// TIA Portal V17 export
// export: Created 2026-04-13T11:12:53.8803486Z, ExportSetting WithDefaults, DisplayName Totally Integrated Automation Portal, DisplayVersion V17 Update 4, DisplayName TIA Portal Openness, DisplayVersion V17 Update 4, DisplayName TIA Portal Version Control Interface, DisplayVersion V17, DisplayName SINAMICS Startdrive Advanced, DisplayVersion V17, DisplayName SINAMICS Startdrive G130, G150, S120, S150, SINAMICS MV, S210, DisplayVersion V17, DisplayName SINAMICS Startdrive G110M, G120, G120C, G120D, G120P, G115D, DisplayVersion V17, DisplayName STEP 7 Professional, DisplayVersion V17 Update 4, DisplayName STEP 7 Safety, DisplayVersion V17, DisplayName WinCC Professional, DisplayVersion V17 Update 4
TagTable "SV"
  SV_BD布袋压差高报 : Real  (PLC tag SV.BD布袋压差高报, HMI_连接_1, 1 s)
  SV_BD布袋压差高高报 : Real  (PLC tag SV.BD布袋压差高高报, HMI_连接_1, 1 s)
  SV_JF进风压差高报 : Real  (PLC tag SV.JF进风压差高报, HMI_连接_1, 1 s)
  SV_JF进风压差高高报 : Real  (PLC tag SV.JF进风压差高高报, HMI_连接_1, 1 s)
  SV_TN塔内压力高高报 : Real  (PLC tag SV.TN塔内压力高高报, HMI_连接_1, 1 s)
  SV_GD管道压力高报 : Real  (PLC tag SV.GD管道压力高报, HMI_连接_1, 1 s)
  SV_GD管道压力高高报 : Real  (PLC tag SV.GD管道压力高高报, HMI_连接_1, 1 s)
  SV_GD管道压力设定 : Real  (PLC tag SV.GD管道压力设定, HMI_连接_1, 1 s)
  SV_TN塔内压力低报 : Real  (PLC tag SV.TN塔内压力低报, HMI_连接_1, 1 s)
  SV_TN塔内压力低低报 : Real  (PLC tag SV.TN塔内压力低低报, HMI_连接_1, 1 s)
  SV_XH循风机频率设定 : Real  (PLC tag SV.XH循风机频率设定, HMI_连接_1, 1 s)
  SV_YF引风频率设定 : Real  (PLC tag SV.YF引风频率设定, HMI_连接_1, 1 s)
  SV_JL进料泵频率设定 : Real  (PLC tag SV.JL进料泵频率设定, HMI_连接_1, 1 s)
  SV_JF进风温度设定 : Real  (PLC tag SV.JF进风温度设定, HMI_连接_1, 1 s)
  SV_CF出温异常设定 : Real  (PLC tag SV.CF出温异常设定, HMI_连接_1, 1 s)
  SV_JF进温高报 : Real  (PLC tag SV.JF进温高报, HMI_连接_1, 1 s)
  SV_JF进温高高报 : Real  (PLC tag SV.JF进温高高报, HMI_连接_1, 1 s)
  SV_CF出风温度设定 : Real  (PLC tag SV.CF出风温度设定, HMI_连接_1, 1 s)
  SV_CF出温高报 : Real  (PLC tag SV.CF出温高报, HMI_连接_1, 1 s)
  SV_CF出温高高报 : Real  (PLC tag SV.CF出温高高报, HMI_连接_1, 1 s)
  SV_WQ尾温高报 : Real  (PLC tag SV.WQ尾温高报, HMI_连接_1, 1 s)
  SV_WQ尾温高高报 : Real  (PLC tag SV.WQ尾温高高报, HMI_连接_1, 1 s)
  SV_BD布袋反吹时间 : Real  (PLC tag SV.BD布袋反吹时间, HMI_连接_1, 1 s)
  SV_TW塔外气锤时间 : Real  (PLC tag SV.TW塔外气锤时间, HMI_连接_1, 1 s)
  SV_TN塔内气扫时间 : Real  (PLC tag SV.TN塔内气扫时间, HMI_连接_1, 1 s)
  SV_DQ氮气下限设定 : Real  (PLC tag SV.DQ氮气下限设定, HMI_连接_1, 1 s)
  SV_TN塔内压力高报 : Real  (PLC tag SV.TN塔内压力高报, HMI_连接_1, 1 s)
  SV_JW降温温度设定 : Real  (PLC tag SV.JW降温温度设定, HMI_连接_1, 1 s)
  SV_LS冷水温度写 : Real  (PLC tag SV.LS冷水温度写, HMI_连接_1, 1 s)
  SV_ZT主塔振打间隔 : Real  (PLC tag SV.ZT主塔振打间隔, HMI_连接_1, 1 s)
  SV_TZ通针时间 : Real  (PLC tag SV.TZ通针时间, HMI_连接_1, 1 s)
  SV_PM屏幕编号 : Real  (PLC tag SV.PM屏幕编号, HMI_连接_1, 1 s)
  SV_YH氧含仪高报 : Real  (PLC tag SV.YH氧含仪高报, HMI_连接_1, 1 s)
  SV_JD进氮压力 : Real  (PLC tag SV.JD进氮压力, HMI_连接_1, 1 s)
  SV_JL进料压力高报 : Real  (PLC tag SV.JL进料压力高报, HMI_连接_1, 1 s)
  SV_JL进料压力高高报 : Real  (PLC tag SV.JL进料压力高高报, HMI_连接_1, 1 s)
  SV_WQ尾气温度 : Real  (PLC tag SV.WQ尾气温度, HMI_连接_1, 1 s)
  SV_JF进风保护温度 : Real  (PLC tag SV.JF进风保护温度, HMI_连接_1, 1 s)
  SV_YH氧含差值 : Real  (PLC tag SV.YH氧含差值, HMI_连接_1, 1 s)
  SV_YH氧含仪1 : Real  (PLC tag SV.YH氧含仪1, HMI_连接_1, 1 s)
  SV_YH氧含仪2 : Real  (PLC tag SV.YH氧含仪2, HMI_连接_1, 1 s)
  SV_LS冷水检测写 : Real  (PLC tag SV.LS冷水检测写, HMI_连接_1, 1 s)
  SV_JF进风检测写 : Real  (PLC tag SV.JF进风检测写, HMI_连接_1, 1 s)
  SV_QT气体检测仪低报 : Real  (PLC tag SV.QT气体检测仪低报, HMI_连接_1, 1 s)
  SV_QT气体检测仪低低报 : Real  (PLC tag SV.QT气体检测仪低低报, HMI_连接_1, 1 s)
  SV_LX离心雾化 : Real  (PLC tag SV.LX离心雾化, HMI_连接_1, 1 s)
  SV_DQ氮气加热写 : Real  (PLC tag SV.DQ氮气加热写, HMI_连接_1, 1 s)
  SV_BD布袋振打时间 : Real  (PLC tag SV.BD布袋振打时间, HMI_连接_1, 1 s)
  SV_PS排水延长时间 : Real  (PLC tag SV.PS排水延长时间, HMI_连接_1, 1 s)
  SV_AQ安全比例阀 : Real  (PLC tag SV.AQ安全比例阀, HMI_连接_1, 1 s)
  SV_PK排空比例阀 : Real  (PLC tag SV.PK排空比例阀, HMI_连接_1, 1 s)
  SV_JB搅拌电机 : Real  (PLC tag SV.JB搅拌电机, HMI_连接_1, 1 s)
  SV_JF进风加热比例调节阀 : Real  (PLC tag SV.JF进风加热比例调节阀, HMI_连接_1, 1 s)
  SV_HF回风加热比例调节阀 : Real  (PLC tag SV.HF回风加热比例调节阀, HMI_连接_1, 1 s)
  SV_FK放空比例调节阀 : Real  (PLC tag SV.FK放空比例调节阀, HMI_连接_1, 1 s)
  SV_SF送风频率 : Real  (PLC tag SV.SF送风频率, HMI_连接_1, 1 s)
  SV_SS输送温度设定 : Real  (PLC tag SV.SS输送温度设定, HMI_连接_1, 1 s)
  SV_BD布袋出料设定 : Real  (PLC tag SV.BD布袋出料设定, HMI_连接_1, 1 s)
  SV_YJ一级旋风出料设定 : Real  (PLC tag SV.YJ一级旋风出料设定, HMI_连接_1, 1 s)
  SV_EJ二级旋风出料设定 : Real  (PLC tag SV.EJ二级旋风出料设定, HMI_连接_1, 1 s)
  SV_BD布袋T出料设定 : Real  (PLC tag SV.BD布袋T出料设定, HMI_连接_1, 1 s)
  SV_YJ一级旋风T出料设定 : Real  (PLC tag SV.YJ一级旋风T出料设定, HMI_连接_1, 1 s)
  SV_EJ二级旋风T出料设定 : Real  (PLC tag SV.EJ二级旋风T出料设定, HMI_连接_1, 1 s)
  SV_BD布袋上阀开时间 : Real  (PLC tag SV.BD布袋上阀开时间, HMI_连接_1, 1 s)
  SV_BD布袋上阀关时间 : Real  (PLC tag SV.BD布袋上阀关时间, HMI_连接_1, 1 s)
  SV_BD布袋下阀开时间 : Real  (PLC tag SV.BD布袋下阀开时间, HMI_连接_1, 1 s)
  SV_BD布袋下阀关时间 : Real  (PLC tag SV.BD布袋下阀关时间, HMI_连接_1, 1 s)
  SV_YJ一级旋风上阀开时间 : Real  (PLC tag SV.YJ一级旋风上阀开时间, HMI_连接_1, 1 s)
  SV_YJ一级旋风上阀关时间 : Real  (PLC tag SV.YJ一级旋风上阀关时间, HMI_连接_1, 1 s)
  SV_YJ一级旋风下阀开时间 : Real  (PLC tag SV.YJ一级旋风下阀开时间, HMI_连接_1, 1 s)
  SV_YJ一级旋风下阀关时间 : Real  (PLC tag SV.YJ一级旋风下阀关时间, HMI_连接_1, 1 s)
  SV_EJ二级旋风上阀开时间 : Real  (PLC tag SV.EJ二级旋风上阀开时间, HMI_连接_1, 1 s)
  SV_EJ二级旋风上阀关时间 : Real  (PLC tag SV.EJ二级旋风上阀关时间, HMI_连接_1, 1 s)
  SV_EJ二级旋风下阀开时间 : Real  (PLC tag SV.EJ二级旋风下阀开时间, HMI_连接_1, 1 s)
  SV_EJ二级旋风下阀关时间 : Real  (PLC tag SV.EJ二级旋风下阀关时间, HMI_连接_1, 1 s)
  SV_HF回风温度设定 : Real  (PLC tag SV.HF回风温度设定, HMI_连接_1, 1 s)
  SV_ZT主塔压力设定 : Real  (PLC tag SV.ZT主塔压力设定, HMI_连接_1, 1 s)
  SV_KQ空气流量设定 : Real  (PLC tag SV.KQ空气流量设定, HMI_连接_1, 1 s)
  SV_JL进料流量设定 : Real  (PLC tag SV.JL进料流量设定, HMI_连接_1, 1 s)
  SV_JL进料泵频率手动设定 : Real  (PLC tag SV.JL进料泵频率手动设定, HMI_连接_1, 1 s)
  SV_YF引风频率手动设定 : Real  (PLC tag SV.YF引风频率手动设定, HMI_连接_1, 1 s)
  SV_JF进风流量设定 : Real  (PLC tag SV.JF进风流量设定, HMI_连接_1, 1 s)
  SV_YF引风频率自动设定 : Real  (PLC tag SV.YF引风频率自动设定, HMI_连接_1, 1 s)
  SV_JL进料频率自动设定 : Real  (PLC tag SV.JL进料频率自动设定, HMI_连接_1, 1 s)
  SV_FD阀导气压低报 : Real  (PLC tag SV.FD阀导气压低报, HMI_连接_1, 1 s)
  SV_FD阀导气压低低报 : Real  (PLC tag SV.FD阀导气压低低报, HMI_连接_1, 1 s)
  SV_JF进风压差低报 : Real  (PLC tag SV.JF进风压差低报, HMI_连接_1, 1 s)
  SV_WH雾化油压低报 : Real  (PLC tag SV.WH雾化油压低报, HMI_连接_1, 1 s)
  SV_WH雾化油压低低报 : Real  (PLC tag SV.WH雾化油压低低报, HMI_连接_1, 1 s)
  SV_JD进氮压力低报 : Real  (PLC tag SV.JD进氮压力低报, HMI_连接_1, 1 s)
  SV_JD进氮压力低低报 : Real  (PLC tag SV.JD进氮压力低低报, HMI_连接_1, 1 s)
  SV_CF出风高效高报 : Real  (PLC tag SV.CF出风高效高报, HMI_连接_1, 1 s)
  SV_CF出风高效高高报 : Real  (PLC tag SV.CF出风高效高高报, HMI_连接_1, 1 s)
  SV_CF出风高效低报 : Real  (PLC tag SV.CF出风高效低报, HMI_连接_1, 1 s)
  SV_SF输送高效高报 : Real  (PLC tag SV.SF输送高效高报, HMI_连接_1, 1 s)
  SV_SF输送高效高高报 : Real  (PLC tag SV.SF输送高效高高报, HMI_连接_1, 1 s)
  SV_SF输送高效低报 : Real  (PLC tag SV.SF输送高效低报, HMI_连接_1, 1 s)
  SV_HF回风温度高报 : Real  (PLC tag SV.HF回风温度高报, HMI_连接_1, 1 s)
  SV_HF回风温度高高报 : Real  (PLC tag SV.HF回风温度高高报, HMI_连接_1, 1 s)
  SV_BD布袋压差低报 : Real  (PLC tag SV.BD布袋压差低报, HMI_连接_1, 1 s)
  SV_SS输送保护温度 : Real  (PLC tag SV.SS输送保护温度, HMI_连接_1, 1 s)
  SV_JL进料停机阈值 : Real  (PLC tag SV.JL进料停机阈值, HMI_连接_1, 1 s)
  SV_SB设备振打间隔 : Real  (PLC tag SV.SB设备振打间隔, HMI_连接_1, 1 s)
  SV_SS输送温度高高报 : Real  (PLC tag SV.SS输送温度高高报, HMI_连接_1, 1 s)
  SV_SS输送温度高报 : Real  (PLC tag SV.SS输送温度高报, HMI_连接_1, 1 s)
  SV_SS输送压差高高报 : Real  (PLC tag SV.SS输送压差高高报, HMI_连接_1, 1 s)
  SV_SS输送压差高报 : Real  (PLC tag SV.SS输送压差高报, HMI_连接_1, 1 s)
  SV_SS输送压差低报 : Real  (PLC tag SV.SS输送压差低报, HMI_连接_1, 1 s)
  SV_YJ一级液位高报 : Real  (PLC tag SV.YJ一级液位高报, HMI_连接_1, 1 s)
  SV_YJ一级液位计高高报 : Real  (PLC tag SV.YJ一级液位计高高报, HMI_连接_1, 1 s)
  SV_EJ二级液位计高报 : Real  (PLC tag SV.EJ二级液位计高报, HMI_连接_1, 1 s)
  SV_EJ二级液位计高高报 : Real  (PLC tag SV.EJ二级液位计高高报, HMI_连接_1, 1 s)
  SV_CW除雾液位计高报 : Real  (PLC tag SV.CW除雾液位计高报, HMI_连接_1, 1 s)
  SV_CW除雾液位计高高报 : Real  (PLC tag SV.CW除雾液位计高高报, HMI_连接_1, 1 s)
  SV_FD阀岛气压低报 : Real  (PLC tag SV.FD阀岛气压低报, HMI_连接_1, 1 s)
  SV_FD阀岛气压低低报 : Real  (PLC tag SV.FD阀岛气压低低报, HMI_连接_1, 1 s)
  SV_YH氧含仪高高报 : Real  (PLC tag SV.YH氧含仪高高报, HMI_连接_1, 1 s)
  SV_JF进风流量低低报 : Real  (PLC tag SV.JF进风流量低低报, HMI_连接_1, 1 s)
  SV_JF进风流量低报 : Real  (PLC tag SV.JF进风流量低报, HMI_连接_1, 1 s)
  SV_QZ前置水罐液位低报 : Real  (PLC tag SV.QZ前置水罐液位低报, HMI_连接_1, 1 s)
  SV_QZ前置水罐液位低低报 : Real  (PLC tag SV.QZ前置水罐液位低低报, HMI_连接_1, 1 s)
  SV_JL进料流量低报 : Real  (PLC tag SV.JL进料流量低报, HMI_连接_1, 1 s)
  SV_JL进料流量低低报 : Real  (PLC tag SV.JL进料流量低低报, HMI_连接_1, 1 s)
  SV_YJ一级旋风振打间隔 : Real  (PLC tag SV.YJ一级旋风振打间隔, HMI_连接_1, 1 s)
  SV_EJ二级旋风振打间隔 : Real  (PLC tag SV.EJ二级旋风振打间隔, HMI_连接_1, 1 s)
  SV_YJ一级旋风振荡运行 : Real  (PLC tag SV.YJ一级旋风振荡运行, HMI_连接_1, 1 s)
  SV_YJ一级旋风振荡停止 : Real  (PLC tag SV.YJ一级旋风振荡停止, HMI_连接_1, 1 s)
  SV_TJ调节单元 : Real  (PLC tag SV.TJ调节单元, HMI_连接_1, 1 s)
  SV_TJ调节时间 : Real  (PLC tag SV.TJ调节时间, HMI_连接_1, 1 s)
  SV_BD布袋压差自动反吹 : Real  (PLC tag SV.BD布袋压差自动反吹, HMI_连接_1, 1 s)
  SV_BD布袋压差自动反吹时间 : Real  (PLC tag SV.BD布袋压差自动反吹时间, HMI_连接_1, 1 s)
  SV_ZT 中途停止温度分界 : Real  (PLC tag SV."ZT 中途停止温度分界", HMI_连接_1, 1 s)
  SV_JX碱洗温度设定 : Real  (PLC tag SV.JX碱洗温度设定, HMI_连接_1, 1 s)
  SV_FK放空阀手动设定 : Real  (PLC tag SV.FK放空阀手动设定, HMI_连接_1, 1 s)
  SV_FK放空阀自动设定 : Real  (PLC tag SV.FK放空阀自动设定, HMI_连接_1, 1 s)
